# EPICS autosave request: LabJackApp/Db/LabJack_binary_settings.req
# Digital input
$(P)Bi$(N).DESC

# Digital output
$(P)Bo$(N).DESC

# Digital direction
$(P)Bd$(N).VAL
